// Mitsubishi GX Works2 project: Pulsado 1 bot   PLC: Q03UDV
// HelloWorld

PROGRAM MAIN
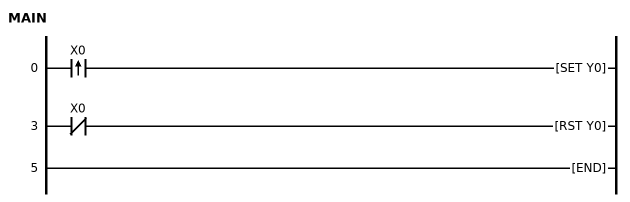
0     LDP     X0
      SET     Y0
3     LDI     X0
      RST     Y0
5     END
END_PROGRAM
